{attribute 'GeneratedUsingTerminal: EQ3204-0002-0021'}
{attribute addProperty BoxType "EQ3204-0002-0021"}
{attribute addProperty Id "RTD_RTDInputs_Channel_1AT %I*RTD_RTDInputs_Channel_4A3944819RTD_RTDInputs_Channel_2AT %I*RTD_RTDInputs_Channel_4A3944819RTD_RTDInputs_Channel_3AT %I*RTD_RTDInputs_Channel_4A3944819RTD_RTDInputs_Channel_4AT %I*RTD_RTDInputs_Channel_4A3944819WcStateAT %I*WcState_9091E0EB2InfoDataAT %I*InfoData_94A18F5E2"}
{attribute addProperty CRC "1540847397"}
{attribute addProperty Size "40"}
TYPE EQ3204_5BD77725 EXTENDS EtcSlaveTerminalBase_947E5A46 :
STRUCT
	{attribute addProperty Name "RTD_RTDInputs_Channel_1"}
	RTD_RTDInputs_Channel_1 : RTD_RTDInputs_Channel_4A394481;
	{attribute addProperty Name "RTD_RTDInputs_Channel_2"}
	RTD_RTDInputs_Channel_2 : RTD_RTDInputs_Channel_4A394481;
	{attribute addProperty Name "RTD_RTDInputs_Channel_3"}
	RTD_RTDInputs_Channel_3 : RTD_RTDInputs_Channel_4A394481;
	{attribute addProperty Name "RTD_RTDInputs_Channel_4"}
	RTD_RTDInputs_Channel_4 : RTD_RTDInputs_Channel_4A394481;
	{attribute addProperty Name "WcState"}
	WcState : WcState_9091E0EB;
	{attribute addProperty Name "InfoData"}
	InfoData : InfoData_94A18F5E;
END_STRUCT
END_TYPE

(* stored: Version 1.2.0.0, ProductVersion 3.1.4024.9
   DUT EQ3204_5BD77725: Id {4cf6a8ca-db80-4e1c-97ca-19fb77a24ac5} *)
